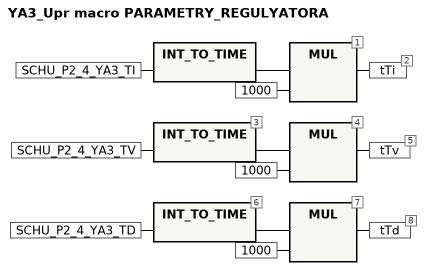
[picture p531: YA3_Upr macro PARAMETRY_REGULYATORA (CFC)]
_CFC_ (* Continuous Function Chart, elements in execution order *)
#0 MACRO PARAMETRY_REGULYATORA()
	#1 INT_TO_TIME(SCHU_P2_4_YA3_TI)
	#2 MUL(#1, 1000)
	#3 tTi <= #2
	#4 INT_TO_TIME(SCHU_P2_4_YA3_TV)
	#5 MUL(#4, 1000)
	#6 tTv <= #5
	#7 INT_TO_TIME(SCHU_P2_4_YA3_TD)
	#8 MUL(#7, 1000)
	#9 tTd <= #8
END_MACRO
#10 AND(SCHU_P2_4_UST_LETO, SCHU_P2_4_UE3_T_DOST, SCHU_P2_4_UST_RE_RABOTA, NOT Z_ZAM_SR, SCHU_P2_4_SA5_DI5_A)
#11 SEL(#10, eHVACCtrlMode_Manual, eHVACCtrlMode_Auto)
#12 OR(SCHU_P2_4_UST_ZIMA, NOT SCHU_P2_4_UST_RE_RABOTA, Z_ZAM_SR)
#13 SEL(#12, SCHU_P2_4_YA3_UP_VN, 0)
#14 SEL(NOT SCHU_P2_4_SA5_DI5_A, #13, SCHU_P2_4_YA3_UP_VN)
#15 MUL(SCHU_P2_4_YA4_ZAD_VN, 0.02)
#16 ADD(SCHU_P2_4_UE3_T_UST, #15)
#17 SUB(SCHU_P2_4_UE3_T_VN, #16)
#18 SUB(SCHU_P2_4_UE3_VL_VN, SCHU_P2_4_UE3_VL_UST)
#19 <(#17, #18)
#20 AND(#19, SCHU_P2_4_UE3_VL_DOST, SCHU_P2_4_UE3_T_DOST)
#21 SEL(#20, #16, SCHU_P2_4_UE3_VL_UST)
#22 SEL(#10, 0, #21)
#23 SEL(#20, SCHU_P2_4_UE3_T_VN, SCHU_P2_4_UE3_VL_VN)
#24 SEL(#10, 0, #23)
#25 YA3_PID:FB_HVACPIDCtrl(eHVACDataSecurityType_Idle, FALSE, TRUE, #22, #24, tTaskCycleTime, tTaskCycleTime, #11, #14, SCHU_P2_4_YA3_UP_VN, FALSE, SCHU_P2_4_SB, deadRange, direction, SCHU_P2_4_YA3_KP, tTi, tTv, tTd, rYMin, rYMax)
#26 SCHU_P2_4_YA3_RASSOG <= #25.out 2
#27 YA3_Otkaz <= #25.out 8
#28 SEL(SCHU_P2_4_SA5_DI5_A, 0, #25.out 1)
#29 SCHU_P2_4_YA3_ZAD_VN <= #28
#30 SUB(#28, SCHU_P2_4_YA3_UP_VN)
#31 SCHU_P2_4_YA3_RASSOG_POL <= #30
_END_CFC_
END_PROGRAM

(* POU IM/YA4_Upr, CFC *)
PROGRAM YA4_Upr
VAR
	YA4_PID: FB_HVACPIDCtrl;

	deadRange: REAL := 0.1;
	direction: BOOL;
	tTi: TIME;
	tTv: TIME;
	tTd: TIME;

	rYMin: REAL := 0;
	rYMax: REAL := 100;
END_VAR
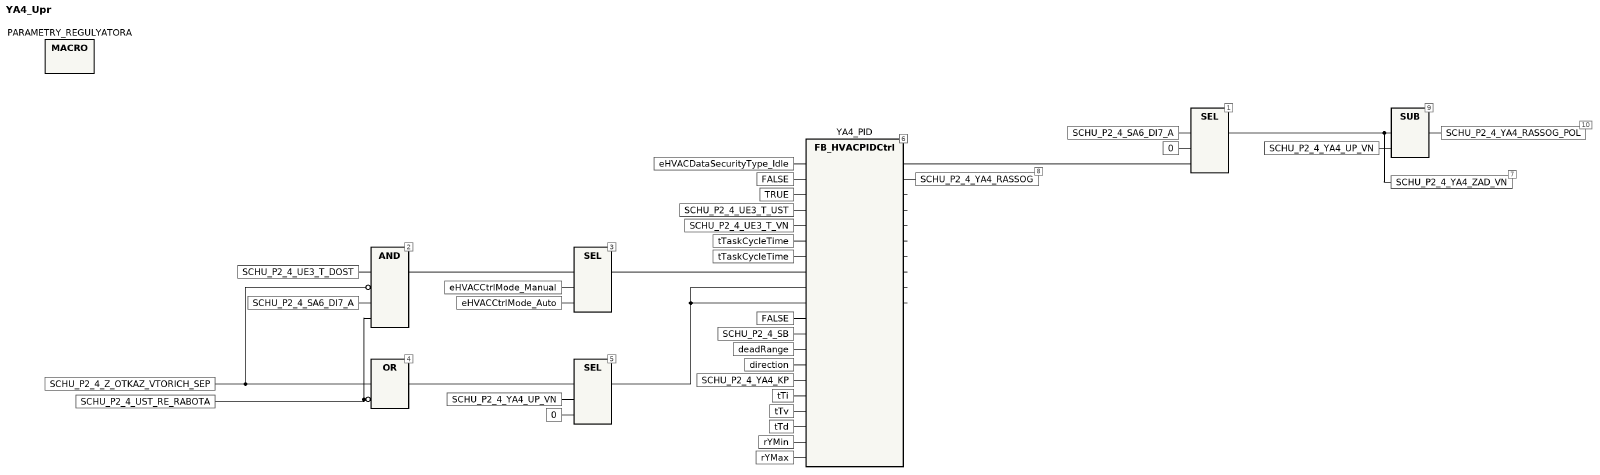
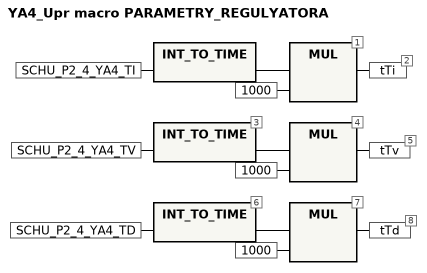
_CFC_ (* Continuous Function Chart, elements in execution order *)
#0 MACRO PARAMETRY_REGULYATORA()
	#1 INT_TO_TIME(SCHU_P2_4_YA4_TI)
	#2 MUL(#1, 1000)
	#3 tTi <= #2
	#4 INT_TO_TIME(SCHU_P2_4_YA4_TV)
	#5 MUL(#4, 1000)
	#6 tTv <= #5
	#7 INT_TO_TIME(SCHU_P2_4_YA4_TD)
	#8 MUL(#7, 1000)
	#9 tTd <= #8
END_MACRO
#10 SEL(SCHU_P2_4_SA6_DI7_A, 0, #15.out 1)
#11 AND(SCHU_P2_4_UE3_T_DOST, NOT SCHU_P2_4_Z_OTKAZ_VTORICH_SEP, SCHU_P2_4_SA6_DI7_A, SCHU_P2_4_UST_RE_RABOTA)
#12 SEL(#11, eHVACCtrlMode_Manual, eHVACCtrlMode_Auto)
#13 OR(SCHU_P2_4_Z_OTKAZ_VTORICH_SEP, NOT SCHU_P2_4_UST_RE_RABOTA)
#14 SEL(#13, SCHU_P2_4_YA4_UP_VN, 0)
#15 YA4_PID:FB_HVACPIDCtrl(eHVACDataSecurityType_Idle, FALSE, TRUE, SCHU_P2_4_UE3_T_UST, SCHU_P2_4_UE3_T_VN, tTaskCycleTime, tTaskCycleTime, #12, #14, #14, FALSE, SCHU_P2_4_SB, deadRange, direction, SCHU_P2_4_YA4_KP, tTi, tTv, tTd, rYMin, rYMax)
#16 SCHU_P2_4_YA4_ZAD_VN <= #10
#17 SCHU_P2_4_YA4_RASSOG <= #15.out 2
#18 SUB(#10, SCHU_P2_4_YA4_UP_VN)
#19 SCHU_P2_4_YA4_RASSOG_POL <= #18
_END_CFC_
END_PROGRAM

(* POU IM/razr_pusk, CFC *)
PROGRAM razr_pusk
VAR
END_VAR
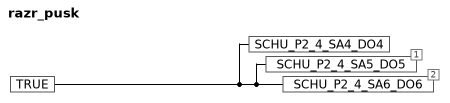
_CFC_ (* Continuous Function Chart, elements in execution order *)
#0 SCHU_P2_4_SA4_DO4 <= TRUE
#1 SCHU_P2_4_SA5_DO5 <= TRUE
#2 SCHU_P2_4_SA6_DO6 <= TRUE
_END_CFC_
(* the same logic as Structured Text *)
SCHU_P2_4_SA4_DO4 := TRUE;
SCHU_P2_4_SA5_DO5 := TRUE;
SCHU_P2_4_SA6_DO6 := TRUE;
END_PROGRAM

(* POU Output/ALL_Output, CFC *)
PROGRAM ALL_Output
VAR
END_VAR
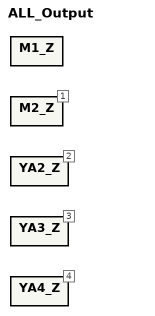
_CFC_ (* Continuous Function Chart, elements in execution order *)
#0 M1_Z()
#1 M2_Z()
#2 YA2_Z()
#3 YA3_Z()
#4 YA4_Z()
_END_CFC_
(* the same logic as Structured Text *)
M1_Z();
M2_Z();
YA2_Z();
YA3_Z();
YA4_Z();
END_PROGRAM

(* POU Output/AO/M1_Z, CFC *)
PROGRAM M1_Z
VAR
	fb_HVACAO_SCHU_P2_4_UZ1_AO1: FB_HVACAnalogOutput;
	enableFeedbCtrl: BOOL := FALSE;
	hysFbCtrl: REAL := 0;
	direction: BOOL;
	delay: TIME := T#0s;
	hi: REAL := 50;
	low: REAL := 0;

END_VAR
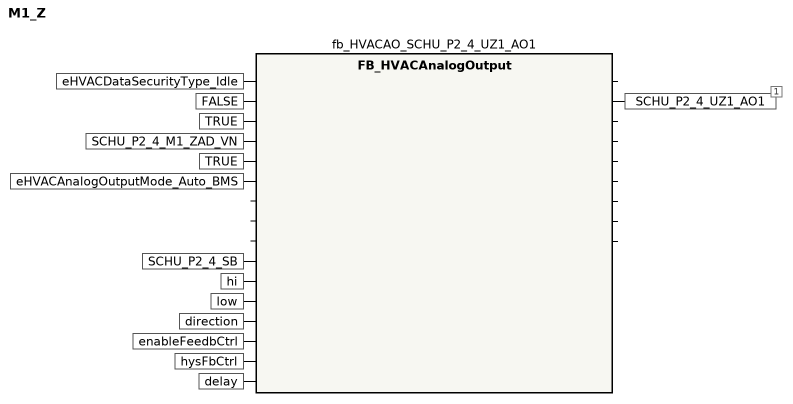
_CFC_ (* Continuous Function Chart, elements in execution order *)
#0 fb_HVACAO_SCHU_P2_4_UZ1_AO1:FB_HVACAnalogOutput(eHVACDataSecurityType_Idle, FALSE, TRUE, SCHU_P2_4_M1_ZAD_VN, TRUE, eHVACAnalogOutputMode_Auto_BMS, -, -, -, SCHU_P2_4_SB, hi, low, direction, enableFeedbCtrl, hysFbCtrl, delay)
#1 SCHU_P2_4_UZ1_AO1 <= #0.out 2
_END_CFC_
END_PROGRAM

(* POU Output/AO/M2_Z, CFC *)
PROGRAM M2_Z
VAR
	fb_HVACAO_SCHU_P2_4_UZ2_AO5: FB_HVACAnalogOutput;
	enableFeedbCtrl: BOOL := FALSE;
	hysFbCtrl: REAL := 0;
	direction: BOOL;
	delay: TIME := T#0s;
	hi: REAL := 50;
	low: REAL := 0;
END_VAR
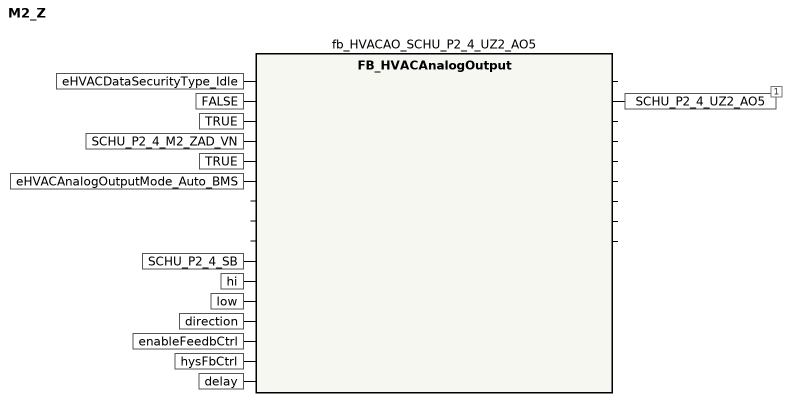
_CFC_ (* Continuous Function Chart, elements in execution order *)
#0 fb_HVACAO_SCHU_P2_4_UZ2_AO5:FB_HVACAnalogOutput(eHVACDataSecurityType_Idle, FALSE, TRUE, SCHU_P2_4_M2_ZAD_VN, TRUE, eHVACAnalogOutputMode_Auto_BMS, -, -, -, SCHU_P2_4_SB, hi, low, direction, enableFeedbCtrl, hysFbCtrl, delay)
#1 SCHU_P2_4_UZ2_AO5 <= #0.out 2
_END_CFC_
END_PROGRAM

(* POU Output/AO/YA2_Z, CFC *)
PROGRAM YA2_Z
VAR
	fb_HVACAO_SCHU_P2_4_YA2_AO2: FB_HVACAnalogOutput;
	enableFeedbCtrl: BOOL := FALSE;
	hysFbCtrl: REAL := 0;
	direction: BOOL;
	delay: TIME := T#0s;
END_VAR
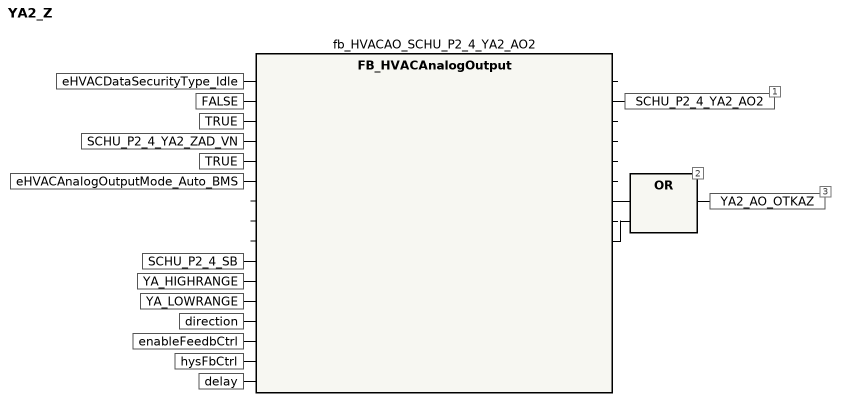
_CFC_ (* Continuous Function Chart, elements in execution order *)
#0 fb_HVACAO_SCHU_P2_4_YA2_AO2:FB_HVACAnalogOutput(eHVACDataSecurityType_Idle, FALSE, TRUE, SCHU_P2_4_YA2_ZAD_VN, TRUE, eHVACAnalogOutputMode_Auto_BMS, -, -, -, SCHU_P2_4_SB, YA_HIGHRANGE, YA_LOWRANGE, direction, enableFeedbCtrl, hysFbCtrl, delay)
#1 SCHU_P2_4_YA2_AO2 <= #0.out 2
#2 OR(#0.out 7, #0.out 9)
#3 YA2_AO_OTKAZ <= #2
_END_CFC_
END_PROGRAM

(* POU Output/AO/YA3_Z, CFC *)
PROGRAM YA3_Z
VAR
	fb_HVACAO_SCHU_P2_4_YA3_AO3: FB_HVACAnalogOutput;
	enableFeedbCtrl: BOOL := FALSE;
	hysFbCtrl: REAL := 0;
	direction: BOOL;
	delay: TIME := T#0s;
END_VAR
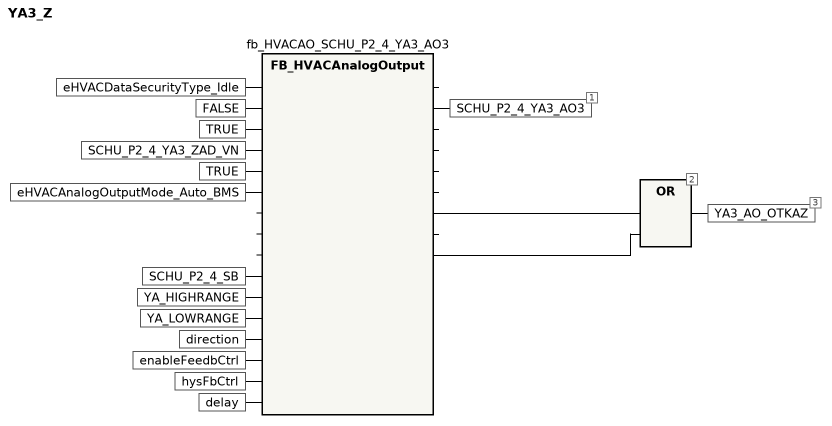
_CFC_ (* Continuous Function Chart, elements in execution order *)
#0 fb_HVACAO_SCHU_P2_4_YA3_AO3:FB_HVACAnalogOutput(eHVACDataSecurityType_Idle, FALSE, TRUE, SCHU_P2_4_YA3_ZAD_VN, TRUE, eHVACAnalogOutputMode_Auto_BMS, -, -, -, SCHU_P2_4_SB, YA_HIGHRANGE, YA_LOWRANGE, direction, enableFeedbCtrl, hysFbCtrl, delay)
#1 SCHU_P2_4_YA3_AO3 <= #0.out 2
#2 OR(#0.out 7, #0.out 9)
#3 YA3_AO_OTKAZ <= #2
_END_CFC_
END_PROGRAM

(* POU Output/AO/YA4_Z, CFC *)
PROGRAM YA4_Z
VAR
	fb_HVACAO_SCHU_P2_4_YA4_AO4: FB_HVACAnalogOutput;
	enableFeedbCtrl: BOOL := FALSE;
	hysFbCtrl: REAL := 0;
	direction: BOOL;
	delay: TIME := T#0s;
END_VAR
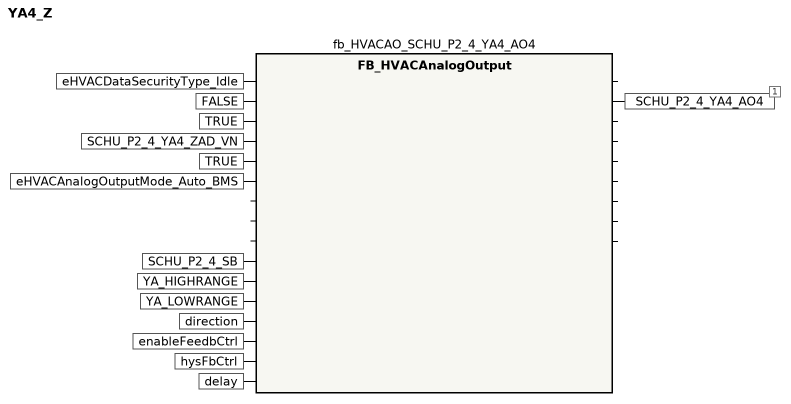
_CFC_ (* Continuous Function Chart, elements in execution order *)
#0 fb_HVACAO_SCHU_P2_4_YA4_AO4:FB_HVACAnalogOutput(eHVACDataSecurityType_Idle, FALSE, TRUE, SCHU_P2_4_YA4_ZAD_VN, TRUE, eHVACAnalogOutputMode_Auto_BMS, -, -, -, SCHU_P2_4_SB, YA_HIGHRANGE, YA_LOWRANGE, direction, enableFeedbCtrl, hysFbCtrl, delay)
#1 SCHU_P2_4_YA4_AO4 <= #0.out 2
_END_CFC_
END_PROGRAM

(* POU Input/ModBus/MB_UZT, CFC *)
PROGRAM MB_UZT
VAR
	MB_READ_REGS: ModbusRtuMaster_KL6x22B;
	Quantity: WORD:= 4;
	MBAddr: WORD:= 16#3000;
	Error: BOOL;
	Errorld: MODBUS_ERRORS;
	cbRead: UINT;

	TON1: TON;

	UnitID_2: BYTE:=2;
	rs_s: RS;
	UnitID_1: BYTE := 1;

	SWT: BOOL;
	ton2: TON;
	tp1: TOF;

END_VAR
